// TIA Portal V16 export
// export: Created 2021-03-04T22:04:04.961948Z, ExportSetting WithDefaults, DisplayName Totally Integrated Automation Portal, DisplayVersion V16, DisplayName TIA Portal Version Control Interface, DisplayVersion V16, DisplayName TIA Portal Openness, DisplayVersion V16, DisplayName SINAMICS Startdrive Advanced, DisplayVersion V16, DisplayName SINAMICS Startdrive G130, G150, S120, S150, SINAMICS MV, S210, DisplayVersion V16, DisplayName SINAMICS Startdrive G110M, G120, G120C, G120D, G120P, DisplayVersion V16, DisplayName STEP 7 Professional, DisplayVersion V16, DisplayName STEP 7 Safety, DisplayVersion V16, DisplayName WinCC Professional, DisplayVersion V16
VAR_GLOBAL   // PLC tag table "System Bits"
   System_Byte AT %MB1 : Byte;   //    {ExternalAccessible false, ExternalVisible false, ExternalWritable false}
   AlwaysFALSE AT %M1.3 : Bool;   //    {ExternalAccessible false, ExternalVisible false, ExternalWritable false}
   "Clock_1.25Hz" AT %M0.4 : Bool;   //    {ExternalAccessible false, ExternalVisible false, ExternalWritable false}
   Clock_1Hz AT %M0.5 : Bool;   //    {ExternalAccessible false, ExternalVisible false, ExternalWritable false}
   "Clock_0.5Hz" AT %M0.7 : Bool;   //    {ExternalAccessible false, ExternalVisible false, ExternalWritable false}
   FirstScan AT %M1.0 : Bool;   //    {ExternalAccessible false, ExternalVisible false, ExternalWritable false}
   Clock_Byte AT %MB0 : Byte;   //    {ExternalAccessible false, ExternalVisible false, ExternalWritable false}
   "Clock_2.5Hz" AT %M0.2 : Bool;   //    {ExternalAccessible false, ExternalVisible false, ExternalWritable false}
   "Clock_0.625Hz" AT %M0.6 : Bool;   //    {ExternalAccessible false, ExternalVisible false, ExternalWritable false}
   Clock_5Hz AT %M0.1 : Bool;   //    {ExternalAccessible false, ExternalVisible false, ExternalWritable false}
   Clock_10Hz AT %M0.0 : Bool;   //    {ExternalAccessible false, ExternalVisible false, ExternalWritable false}
   AlwaysTRUE AT %M1.2 : Bool;   //    {ExternalAccessible false, ExternalVisible false, ExternalWritable false}
   DiagStatusUpdate AT %M1.1 : Bool;   //    {ExternalAccessible false, ExternalVisible false, ExternalWritable false}
   Clock_2Hz AT %M0.3 : Bool;   //    {ExternalAccessible false, ExternalVisible false, ExternalWritable false}
END_VAR
